LIN {X 0,Y 90.441,Z 484.223,A -85,B 0,C 180,E1 -28590.27,E2 -28590.27} C_VEL
LIN {X 0,Y 89.937,Z 477.189,A -85,B 0,C 180,E1 -28595.779,E2 -28595.779} C_VEL
LIN {X 0,Y 88.998,Z 470.496,A -85,B 0,C 180,E1 -28601.586,E2 -28601.586} C_VEL
LIN {X 0,Y 88.423,Z 466.907,A -85,B 0,C 180,E1 -28605.03,E2 -28605.03} C_VEL
LIN {X 0,Y 87.757,Z 463.816,A -85,B 0,C 180,E1 -28608.45,E2 -28608.45} C_VEL
LIN {X 0,Y 86.788,Z 460.611,A -85,B 0,C 180,E1 -28613.023,E2 -28613.023} C_VEL
LIN {X 0,Y 85.348,Z 457.502,A -85,B 0,C 180,E1 -28620,E2 -28620} C_VEL
LIN {X 0,Y 84.954,Z 455.593,A -85,B 0,C 180,E1 -28624.745,E2 -28624.745} C_VEL
LIN {X 0,Y 84.227,Z 455.367,A -85,B 0,C 180,E1 -28634.496,E2 -28634.496} C_VEL
LIN {X 0,Y 84.372,Z 456.038,A -85,B 0,C 180,E1 -28639.462,E2 -28639.462} C_VEL
LIN {X 0,Y 85.474,Z 459.487,A -85,B 0,C 180,E1 -28649.56,E2 -28649.56} C_VEL
LIN {X 0,Y 87.06,Z 463.676,A -85,B 0,C 180,E1 -28657.257,E2 -28657.257} C_VEL
LIN {X 0,Y 88.372,Z 467.412,A -85,B 0,C 180,E1 -28662.533,E2 -28662.533} C_VEL
LIN {X 0,Y 89.775,Z 472.169,A -85,B 0,C 180,E1 -28668.124,E2 -28668.124} C_VEL
LIN {X 0,Y 90.788,Z 476.909,A -85,B 0,C 180,E1 -28672.909,E2 -28672.909} C_VEL
LIN {X 0,Y 91.718,Z 483.277,A -85,B 0,C 180,E1 -28678.72,E2 -28678.72} C_VEL
LIN {X 0,Y 91.813,Z 484.853,A -85,B 0,C 180,E1 -28680.112,E2 -28680.112} C_VEL
LIN {X 0,Y 91.514,Z 486.512,A -85,B 0,C 180,E1 -28681.287,E2 -28681.287} C_VEL
LIN {X 0,Y 85.387,Z 495.474,A -85,B 0,C 180,E1 -28685.689,E2 -28685.689} C_VEL
LIN {X 0,Y 78.734,Z 504.116,A -85,B 0,C 180,E1 -28691.785,E2 -28691.785} C_VEL
LIN {X 0,Y 73.023,Z 511.07,A -85,B 0,C 180,E1 -28698.891,E2 -28698.891} C_VEL
LIN {X 0,Y 68.391,Z 516.618,A -85,B 0,C 180,E1 -28707.044,E2 -28707.044} C_VEL
LIN {X 0,Y 65.021,Z 520.925,A -85,B 0,C 180,E1 -28716.193,E2 -28716.193} C_VEL
LIN {X 0,Y 63.992,Z 522.397,A -85,B 0,C 180,E1 -28720.372,E2 -28720.372} C_VEL
LIN {X 0,Y 62.488,Z 523.952,A -85,B 0,C 180,E1 -28725.374,E2 -28725.374} C_VEL
LIN {X 0,Y 59.217,Z 525.988,A -85,B 0,C 180,E1 -28734.001,E2 -28734.001} C_VEL
LIN {X 0,Y 57.425,Z 527.14,A -85,B 0,C 180,E1 -28741.567,E2 -28741.567} C_VEL
LIN {X 0,Y 57.494,Z 527.667,A -85,B 0,C 180,E1 -28747.475,E2 -28747.475} C_VEL
LIN {X 0,Y 57.899,Z 527.754,A -85,B 0,C 180,E1 -28749.398,E2 -28749.398} C_VEL
LIN {X 0,Y 59.806,Z 527.977,A -85,B 0,C 180,E1 -28755.165,E2 -28755.165} C_VEL
LIN {X 0,Y 62.746,Z 527.792,A -85,B 0,C 180,E1 -28761.611,E2 -28761.611} C_VEL
LIN {X 0,Y 66.995,Z 527.076,A -85,B 0,C 180,E1 -28768.365,E2 -28768.365} C_VEL
LIN {X 0,Y 70.922,Z 526.057,A -85,B 0,C 180,E1 -28773.081,E2 -28773.081} C_VEL
LIN {X 0,Y 76.45,Z 524.23,A -85,B 0,C 180,E1 -28778.426,E2 -28778.426} C_VEL
LIN {X 0,Y 84.043,Z 521.069,A -85,B 0,C 180,E1 -28784.048,E2 -28784.048} C_VEL
LIN {X 0,Y 93.053,Z 516.427,A -85,B 0,C 180,E1 -28789.016,E2 -28789.016} C_VEL
LIN {X 0,Y 102.281,Z 510.549,A -85,B 0,C 180,E1 -28793.037,E2 -28793.037} C_VEL
LIN {X 0,Y 103.385,Z 509.573,A -85,B 0,C 180,E1 -28794.148,E2 -28794.148} C_VEL
LIN {X 0,Y 104.857,Z 507.368,A -85,B 0,C 180,E1 -28800,E2 -28800} C_VEL
LIN {X 0,Y 105.694,Z 506.321,A -85,B 0,C 180,E1 -28804.242,E2 -28804.242} C_VEL
LIN {X 0,Y 105.435,Z 506.439,A -85,B 0,C 180,E1 -28807.662,E2 -28807.662} C_VEL
LIN {X 0,Y 104.952,Z 507.069,A -85,B 0,C 180,E1 -28811.589,E2 -28811.589} C_VEL
LIN {X 0,Y 104.419,Z 508.123,A -85,B 0,C 180,E1 -28815.618,E2 -28815.618} C_VEL
LIN {X 0,Y 103.533,Z 509.855,A -85,B 0,C 180,E1 -28819.841,E2 -28819.841} C_VEL
LIN {X 0,Y 101.953,Z 512.493,A -85,B 0,C 180,E1 -28824.432,E2 -28824.432} C_VEL
LIN {X 0,Y 101.315,Z 513.342,A -85,B 0,C 180,E1 -28825.627,E2 -28825.627} C_VEL
LIN {X 0,Y 96.268,Z 517.412,A -85,B 0,C 180,E1 -28828.849,E2 -28828.849} C_VEL
LIN {X 0,Y 87.845,Z 522.625,A -85,B 0,C 180,E1 -28832.873,E2 -28832.873} C_VEL
LIN {X 0,Y 79.912,Z 526.75,A -85,B 0,C 180,E1 -28837.689,E2 -28837.689} C_VEL
LIN {X 0,Y 75.036,Z 528.969,A -85,B 0,C 180,E1 -28841.487,E2 -28841.487} C_VEL
LIN {X 0,Y 66.422,Z 532.14,A -85,B 0,C 180,E1 -28850.607,E2 -28850.607} C_VEL
LIN {X 0,Y 59.941,Z 533.826,A -85,B 0,C 180,E1 -28862.046,E2 -28862.046} C_VEL
LIN {X 0,Y 56.515,Z 533.981,A -85,B 0,C 180,E1 -28875.613,E2 -28875.613} C_VEL
LIN {X 0,Y 55.964,Z 533.494,A -85,B 0,C 180,E1 -28882.8,E2 -28882.8} C_VEL
LIN {X 0,Y 56.103,Z 532.623,A -85,B 0,C 180,E1 -28890.014,E2 -28890.014} C_VEL
LIN {X 0,Y 56.014,Z 531.262,A -85,B 0,C 180,E1 -28897.222,E2 -28897.222} C_VEL
LIN {X 0,Y 57.203,Z 528.349,A -85,B 0,C 180,E1 -28907.902,E2 -28907.902} C_VEL
LIN {X 0,Y 60.084,Z 524.365,A -85,B 0,C 180,E1 -28917.91,E2 -28917.91} C_VEL
LIN {X 0,Y 65.45,Z 518.205,A -85,B 0,C 180,E1 -28928.143,E2 -28928.143} C_VEL
LIN {X 0,Y 71.779,Z 510.926,A -85,B 0,C 180,E1 -28936.081,E2 -28936.081} C_VEL
LIN {X 0,Y 77.139,Z 504.599,A -85,B 0,C 180,E1 -28940.762,E2 -28940.762} C_VEL
LIN {X 0,Y 80.643,Z 497.54,A -85,B 0,C 180,E1 -28945.901,E2 -28945.901} C_VEL
LIN {X 0,Y 84.079,Z 489.495,A -85,B 0,C 180,E1 -28950.853,E2 -28950.853} C_VEL
LIN {X 0,Y 84.644,Z 487.711,A -85,B 0,C 180,E1 -28951.95,E2 -28951.95} C_VEL
LIN {X 0,Y 84.762,Z 482.126,A -85,B 0,C 180,E1 -28956.675,E2 -28956.675} C_VEL
LIN {X 0,Y 84.327,Z 475.376,A -85,B 0,C 180,E1 -28963.04,E2 -28963.04} C_VEL
LIN {X 0,Y 84.038,Z 471.877,A -85,B 0,C 180,E1 -28966.704,E2 -28966.704} C_VEL
LIN {X 0,Y 83.62,Z 468.911,A -85,B 0,C 180,E1 -28970.323,E2 -28970.323} C_VEL
LIN {X 0,Y 82.89,Z 465.961,A -85,B 0,C 180,E1 -28975.136,E2 -28975.136} C_VEL
LIN {X 0,Y 81.806,Z 462.103,A -85,B 0,C 180,E1 -28984.928,E2 -28984.928} C_VEL
LIN {X 0,Y 81.308,Z 461.735,A -85,B 0,C 180,E1 -28989.955,E2 -28989.955} C_VEL
LIN {X 0,Y 81.14,Z 461.858,A -85,B 0,C 180,E1 -28995.061,E2 -28995.061} C_VEL
LIN {X 0,Y 81.15,Z 462.183,A -85,B 0,C 180,E1 -28997.675,E2 -28997.675} C_VEL
LIN {X 0,Y 81.373,Z 464.57,A -85,B 0,C 180,E1 -29005.584,E2 -29005.584} C_VEL
LIN {X 0,Y 82.082,Z 466.661,A -85,B 0,C 180,E1 -29011.089,E2 -29011.089} C_VEL
LIN {X 0,Y 82.948,Z 469.361,A -85,B 0,C 180,E1 -29016.377,E2 -29016.377} C_VEL
LIN {X 0,Y 84.19,Z 474.136,A -85,B 0,C 180,E1 -29023.498,E2 -29023.498} C_VEL
LIN {X 0,Y 85.05,Z 478.302,A -85,B 0,C 180,E1 -29028.607,E2 -29028.607} C_VEL
LIN {X 0,Y 85.741,Z 484.381,A -85,B 0,C 180,E1 -29035.052,E2 -29035.052} C_VEL
LIN {X 0,Y 85.877,Z 486.915,A -85,B 0,C 180,E1 -29037.587,E2 -29037.587} C_VEL
LIN {X 0,Y 85.271,Z 488.72,A -85,B 0,C 180,E1 -29038.852,E2 -29038.852} C_VEL
LIN {X 0,Y 78.274,Z 498.056,A -85,B 0,C 180,E1 -29043.879,E2 -29043.879} C_VEL
LIN {X 0,Y 71.751,Z 505.832,A -85,B 0,C 180,E1 -29049.94,E2 -29049.94} C_VEL
LIN {X 0,Y 65.785,Z 512.512,A -85,B 0,C 180,E1 -29057.651,E2 -29057.651} C_VEL
LIN {X 0,Y 60.935,Z 517.82,A -85,B 0,C 180,E1 -29066.681,E2 -29066.681} C_VEL
LIN {X 0,Y 57.053,Z 522.583,A -85,B 0,C 180,E1 -29079.022,E2 -29079.022} C_VEL
LIN {X 0,Y 55.679,Z 525.751,A -85,B 0,C 180,E1 -29092.236,E2 -29092.236} C_VEL
LIN {X 0,Y 56.136,Z 526.928,A -85,B 0,C 180,E1 -29100.035,E2 -29100.035} C_VEL
LIN {X 0,Y 57.899,Z 527.754,A -85,B 0,C 180,E1 -29109.398,E2 -29109.398} C_VEL
LIN {X 0,Y 59.042,Z 528.024,A -85,B 0,C 180,E1 -29115.071,E2 -29115.071} C_VEL
LIN {X 0,Y 60.377,Z 527.97,A -85,B 0,C 180,E1 -29124.505,E2 -29124.505} C_VEL
LIN {X 0,Y 62.37,Z 527.54,A -85,B 0,C 180,E1 -29131.69,E2 -29131.69} C_VEL
LIN {X 0,Y 65.1,Z 526.861,A -85,B 0,C 180,E1 -29136.377,E2 -29136.377} C_VEL
LIN {X 0,Y 66.308,Z 526.494,A -85,B 0,C 180,E1 -29137.716,E2 -29137.716} C_VEL
LIN {X 0,Y 76.139,Z 523.39,A -85,B 0,C 180,E1 -29145.696,E2 -29145.696} C_VEL
LIN {X 0,Y 85.388,Z 519.424,A -85,B 0,C 180,E1 -29150.934,E2 -29150.934} C_VEL
LIN {X 0,Y 94.427,Z 514.574,A -85,B 0,C 180,E1 -29154.868,E2 -29154.868} C_VEL
LIN {X 0,Y 97.002,Z 512.984,A -85,B 0,C 180,E1 -29155.846,E2 -29155.846} C_VEL
LIN {X 0,Y 98.399,Z 511.735,A -85,B 0,C 180,E1 -29158.778,E2 -29158.778} C_VEL
LIN {X 0,Y 99.81,Z 510.338,A -85,B 0,C 180,E1 -29164.038,E2 -29164.038} C_VEL
LIN {X 0,Y 99.426,Z 510.581,A -85,B 0,C 180,E1 -29168.334,E2 -29168.334} C_VEL
LIN {X 0,Y 98.88,Z 511.281,A -85,B 0,C 180,E1 -29172.312,E2 -29172.312} C_VEL
LIN {X 0,Y 98.084,Z 512.526,A -85,B 0,C 180,E1 -29176.656,E2 -29176.656} C_VEL
LIN {X 0,Y 96.683,Z 514.564,A -85,B 0,C 180,E1 -29181.313,E2 -29181.313} C_VEL
LIN {X 0,Y 95.153,Z 516.094,A -85,B 0,C 180,E1 -29183.597,E2 -29183.597} C_VEL
LIN {X 0,Y 90.116,Z 519.454,A -85,B 0,C 180,E1 -29186.273,E2 -29186.273} C_VEL
LIN {X 0,Y 81.309,Z 524.147,A -85,B 0,C 180,E1 -29190.212,E2 -29190.212} C_VEL
LIN {X 0,Y 72.777,Z 527.943,A -85,B 0,C 180,E1 -29195.41,E2 -29195.41} C_VEL
LIN {X 0,Y 65.575,Z 530.553,A -85,B 0,C 180,E1 -29201.409,E2 -29201.409} C_VEL
LIN {X 0,Y 57.067,Z 532.862,A -85,B 0,C 180,E1 -29212.01,E2 -29212.01} C_VEL
LIN {X 0,Y 51.27,Z 533.634,A -85,B 0,C 180,E1 -29225.735,E2 -29225.735} C_VEL
LIN {X 0,Y 48.918,Z 532.935,A -85,B 0,C 180,E1 -29241.756,E2 -29241.756} C_VEL
LIN {X 0,Y 49.001,Z 532.012,A -85,B 0,C 180,E1 -29250.016,E2 -29250.016} C_VEL
LIN {X 0,Y 48.962,Z 530.551,A -85,B 0,C 180,E1 -29258.268,E2 -29258.268} C_VEL
LIN {X 0,Y 50.484,Z 527.539,A -85,B 0,C 180,E1 -29270.383,E2 -29270.383} C_VEL
LIN {X 0,Y 53.89,Z 523.437,A -85,B 0,C 180,E1 -29281.459,E2 -29281.459} C_VEL
LIN {X 0,Y 59.997,Z 517.137,A -85,B 0,C 180,E1 -29292.358,E2 -29292.358} C_VEL
LIN {X 0,Y 66.782,Z 509.967,A -85,B 0,C 180,E1 -29300.253,E2 -29300.253} C_VEL
LIN {X 0,Y 71.53,Z 504.715,A -85,B 0,C 180,E1 -29304.17,E2 -29304.17} C_VEL
LIN {X 0,Y 75.432,Z 497.757,A -85,B 0,C 180,E1 -29309.54,E2 -29309.54} C_VEL
LIN {X 0,Y 78.485,Z 491.588,A -85,B 0,C 180,E1 -29313.587,E2 -29313.587} C_VEL
LIN {X 0,Y 79.11,Z 489.992,A -85,B 0,C 180,E1 -29314.678,E2 -29314.678} C_VEL
LIN {X 0,Y 79.448,Z 483.823,A -85,B 0,C 180,E1 -29320.626,E2 -29320.626} C_VEL
LIN {X 0,Y 79.489,Z 478.327,A -85,B 0,C 180,E1 -29326.583,E2 -29326.583} C_VEL
LIN {X 0,Y 79.317,Z 473.834,A -85,B 0,C 180,E1 -29332.362,E2 -29332.362} C_VEL
LIN {X 0,Y 79.094,Z 472.344,A -85,B 0,C 180,E1 -29334.902,E2 -29334.902} C_VEL
LIN {X 0,Y 78.327,Z 468.39,A -85,B 0,C 180,E1 -29345.147,E2 -29345.147} C_VEL
LIN {X 0,Y 77.89,Z 467.98,A -85,B 0,C 180,E1 -29350.396,E2 -29350.396} C_VEL
LIN {X 0,Y 77.71,Z 468.178,A -85,B 0,C 180,E1 -29355.742,E2 -29355.742} C_VEL
LIN {X 0,Y 77.625,Z 470.599,A -85,B 0,C 180,E1 -29365.104,E2 -29365.104} C_VEL
LIN {X 0,Y 78.239,Z 473.491,A -85,B 0,C 180,E1 -29372.613,E2 -29372.613} C_VEL
LIN {X 0,Y 78.927,Z 476.658,A -85,B 0,C 180,E1 -29378.558,E2 -29378.558} C_VEL
LIN {X 0,Y 79.612,Z 480.989,A -85,B 0,C 180,E1 -29385.059,E2 -29385.059} C_VEL
LIN {X 0,Y 79.935,Z 485.011,A -85,B 0,C 180,E1 -29390.085,E2 -29390.085} C_VEL
LIN {X 0,Y 80.042,Z 489.079,A -85,B 0,C 180,E1 -29394.822,E2 -29394.822} C_VEL
LIN {X 0,Y 79.105,Z 490.913,A -85,B 0,C 180,E1 -29396.076,E2 -29396.076} C_VEL
LIN {X 0,Y 72.231,Z 499.397,A -85,B 0,C 180,E1 -29400.878,E2 -29400.878} C_VEL
LIN {X 0,Y 64.894,Z 507.442,A -85,B 0,C 180,E1 -29407.713,E2 -29407.713} C_VEL
LIN {X 0,Y 58.526,Z 513.89,A -85,B 0,C 180,E1 -29416.09,E2 -29416.09} C_VEL
LIN {X 0,Y 53.476,Z 519.006,A -85,B 0,C 180,E1 -29426.218,E2 -29426.218} C_VEL
LIN {X 0,Y 49.813,Z 523.223,A -85,B 0,C 180,E1 -29439.028,E2 -29439.028} C_VEL
LIN {X 0,Y 48.789,Z 524.988,A -85,B 0,C 180,E1 -29446.727,E2 -29446.727} C_VEL
LIN {X 0,Y 49.083,Z 527.2,A -85,B 0,C 180,E1 -29460.784,E2 -29460.784} C_VEL
LIN {X 0,Y 51.529,Z 528.252,A -85,B 0,C 180,E1 -29472.974,E2 -29472.974} C_VEL
LIN {X 0,Y 54.458,Z 528.412,A -85,B 0,C 180,E1 -29480.72,E2 -29480.72} C_VEL
LIN {X 0,Y 58.189,Z 528.147,A -85,B 0,C 180,E1 -29487.693,E2 -29487.693} C_VEL
LIN {X 0,Y 62.669,Z 527.402,A -85,B 0,C 180,E1 -29493.757,E2 -29493.757} C_VEL
LIN {X 0,Y 66.308,Z 526.494,A -85,B 0,C 180,E1 -29497.716,E2 -29497.716} C_VEL
LIN {X 0,Y 69.792,Z 525.541,A -85,B 0,C 180,E1 -29501.66,E2 -29501.66} C_VEL
LIN {X 0,Y 74.846,Z 523.681,A -85,B 0,C 180,E1 -29508.271,E2 -29508.271} C_VEL
LIN {X 0,Y 80.569,Z 521.096,A -85,B 0,C 180,E1 -29513.925,E2 -29513.925} C_VEL
LIN {X 0,Y 84.857,Z 519.007,A -85,B 0,C 180,E1 -29516.331,E2 -29516.331} C_VEL
LIN {X 0,Y 91.37,Z 515.634,A -85,B 0,C 180,E1 -29518.767,E2 -29518.767} C_VEL
LIN {X 0,Y 92.402,Z 514.992,A -85,B 0,C 180,E1 -29520,E2 -29520} C_VEL
LIN {X 0,Y 93.655,Z 514.058,A -85,B 0,C 180,E1 -29524.304,E2 -29524.304} C_VEL
LIN {X 0,Y 93.23,Z 514.366,A -85,B 0,C 180,E1 -29528.672,E2 -29528.672} C_VEL
LIN {X 0,Y 92.462,Z 515.24,A -85,B 0,C 180,E1 -29533.181,E2 -29533.181} C_VEL
LIN {X 0,Y 91.316,Z 516.685,A -85,B 0,C 180,E1 -29537.93,E2 -29537.93} C_VEL
LIN {X 0,Y 90.045,Z 517.894,A -85,B 0,C 180,E1 -29540.539,E2 -29540.539} C_VEL
LIN {X 0,Y 87.167,Z 519.66,A -85,B 0,C 180,E1 -29542.024,E2 -29542.024} C_VEL
LIN {X 0,Y 77.972,Z 524.22,A -85,B 0,C 180,E1 -29545.689,E2 -29545.689} C_VEL
LIN {X 0,Y 66.437,Z 528.712,A -85,B 0,C 180,E1 -29552.215,E2 -29552.215} C_VEL
LIN {X 0,Y 56.114,Z 531.645,A -85,B 0,C 180,E1 -29561.304,E2 -29561.304} C_VEL
LIN {X 0,Y 47.795,Z 533.023,A -85,B 0,C 180,E1 -29573.993,E2 -29573.993} C_VEL
LIN {X 0,Y 42.863,Z 532.952,A -85,B 0,C 180,E1 -29590.877,E2 -29590.877} C_VEL
LIN {X 0,Y 41.913,Z 532.367,A -85,B 0,C 180,E1 -29600.366,E2 -29600.366} C_VEL
LIN {X 0,Y 41.909,Z 531.355,A -85,B 0,C 180,E1 -29610.018,E2 -29610.018} C_VEL
LIN {X 0,Y 41.954,Z 529.828,A -85,B 0,C 180,E1 -29619.662,E2 -29619.662} C_VEL
LIN {X 0,Y 43.864,Z 526.7,A -85,B 0,C 180,E1 -29633.632,E2 -29633.632} C_VEL
LIN {X 0,Y 47.938,Z 522.479,A -85,B 0,C 180,E1 -29645.923,E2 -29645.923} C_VEL
LIN {X 0,Y 54.937,Z 516.055,A -85,B 0,C 180,E1 -29657.377,E2 -29657.377} C_VEL
LIN {X 0,Y 62.198,Z 508.957,A -85,B 0,C 180,E1 -29665.066,E2 -29665.066} C_VEL
LIN {X 0,Y 66.212,Z 504.813,A -85,B 0,C 180,E1 -29668.14,E2 -29668.14} C_VEL
LIN {X 0,Y 70.548,Z 497.906,A -85,B 0,C 180,E1 -29673.734,E2 -29673.734} C_VEL
LIN {X 0,Y 73.544,Z 492.433,A -85,B 0,C 180,E1 -29677.527,E2 -29677.527} C_VEL
LIN {X 0,Y 74.259,Z 486.999,A -85,B 0,C 180,E1 -29683.505,E2 -29683.505} C_VEL
LIN {X 0,Y 74.712,Z 482.326,A -85,B 0,C 180,E1 -29689.155,E2 -29689.155} C_VEL
LIN {X 0,Y 74.871,Z 478.616,A -85,B 0,C 180,E1 -29694.613,E2 -29694.613} C_VEL
LIN {X 0,Y 74.578,Z 476.29,A -85,B 0,C 180,E1 -29700,E2 -29700} C_VEL
LIN {X 0,Y 74.428,Z 474.435,A -85,B 0,C 180,E1 -29705.955,E2 -29705.955} C_VEL
LIN {X 0,Y 74.119,Z 474.05,A -85,B 0,C 180,E1 -29710.931,E2 -29710.931} C_VEL
LIN {X 0,Y 73.723,Z 474.655,A -85,B 0,C 180,E1 -29717.549,E2 -29717.549} C_VEL
LIN {X 0,Y 73.548,Z 475.826,A -85,B 0,C 180,E1 -29722.471,E2 -29722.471} C_VEL
LIN {X 0,Y 73.794,Z 478.622,A -85,B 0,C 180,E1 -29730.984,E2 -29730.984} C_VEL
LIN {X 0,Y 74.109,Z 481.26,A -85,B 0,C 180,E1 -29736.587,E2 -29736.587} C_VEL
LIN {X 0,Y 74.396,Z 485.323,A -85,B 0,C 180,E1 -29743.47,E2 -29743.47} C_VEL
LIN {X 0,Y 74.358,Z 489.359,A -85,B 0,C 180,E1 -29749.123,E2 -29749.123} C_VEL
LIN {X 0,Y 74.27,Z 491.359,A -85,B 0,C 180,E1 -29751.771,E2 -29751.771} C_VEL
LIN {X 0,Y 73.025,Z 493.187,A -85,B 0,C 180,E1 -29752.88,E2 -29752.88} C_VEL
LIN {X 0,Y 65.9,Z 501.232,A -85,B 0,C 180,E1 -29757.763,E2 -29757.763} C_VEL
LIN {X 0,Y 58.105,Z 509.001,A -85,B 0,C 180,E1 -29764.94,E2 -29764.94} C_VEL
LIN {X 0,Y 51.021,Z 515.533,A -85,B 0,C 180,E1 -29774.628,E2 -29774.628} C_VEL
LIN {X 0,Y 45.965,Z 520.168,A -85,B 0,C 180,E1 -29785.599,E2 -29785.599} C_VEL
LIN {X 0,Y 42.483,Z 523.933,A -85,B 0,C 180,E1 -29799.504,E2 -29799.504} C_VEL
LIN {X 0,Y 41.545,Z 525.813,A -85,B 0,C 180,E1 -29809.755,E2 -29809.755} C_VEL
LIN {X 0,Y 42.27,Z 527.651,A -85,B 0,C 180,E1 -29823.767,E2 -29823.767} C_VEL
LIN {X 0,Y 46.144,Z 528.766,A -85,B 0,C 180,E1 -29839.572,E2 -29839.572} C_VEL
LIN {X 0,Y 49.867,Z 528.849,A -85,B 0,C 180,E1 -29847.706,E2 -29847.706} C_VEL
LIN {X 0,Y 57.68,Z 527.984,A -85,B 0,C 180,E1 -29858.56,E2 -29858.56} C_VEL
LIN {X 0,Y 65.306,Z 526.283,A -85,B 0,C 180,E1 -29865.539,E2 -29865.539} C_VEL
LIN {X 0,Y 74.584,Z 523.35,A -85,B 0,C 180,E1 -29871.576,E2 -29871.576} C_VEL
LIN {X 0,Y 84.857,Z 519.007,A -85,B 0,C 180,E1 -29876.331,E2 -29876.331} C_VEL
LIN {X 0,Y 86.147,Z 518.315,A -85,B 0,C 180,E1 -29877.489,E2 -29877.489} C_VEL
LIN {X 0,Y 86.682,Z 517.932,A -85,B 0,C 180,E1 -29879.492,E2 -29879.492} C_VEL
LIN {X 0,Y 86.971,Z 517.633,A -85,B 0,C 180,E1 -29883.597,E2 -29883.597} C_VEL
LIN {X 0,Y 87.316,Z 517.45,A -85,B 0,C 180,E1 -29884.617,E2 -29884.617} C_VEL
LIN {X 0,Y 86.809,Z 517.845,A -85,B 0,C 180,E1 -29889.319,E2 -29889.319} C_VEL
LIN {X 0,Y 86.268,Z 518.381,A -85,B 0,C 180,E1 -29892.195,E2 -29892.195} C_VEL
LIN {X 0,Y 85.66,Z 518.923,A -85,B 0,C 180,E1 -29894.249,E2 -29894.249} C_VEL
LIN {X 0,Y 84.135,Z 520.127,A -85,B 0,C 180,E1 -29897.684,E2 -29897.684} C_VEL
LIN {X 0,Y 72.028,Z 525.5,A -85,B 0,C 180,E1 -29902.068,E2 -29902.068} C_VEL
LIN {X 0,Y 62.918,Z 528.601,A -85,B 0,C 180,E1 -29906.7,E2 -29906.7} C_VEL
LIN {X 0,Y 57.16,Z 530.193,A -85,B 0,C 180,E1 -29910.637,E2 -29910.637} C_VEL
LIN {X 0,Y 46.662,Z 532.173,A -85,B 0,C 180,E1 -29921.169,E2 -29921.169} C_VEL
LIN {X 0,Y 38.696,Z 532.705,A -85,B 0,C 180,E1 -29937.009,E2 -29937.009} C_VEL
LIN {X 0,Y 36.201,Z 532.434,A -85,B 0,C 180,E1 -29947.176,E2 -29947.176} C_VEL
LIN {X 0,Y 34.923,Z 531.758,A -85,B 0,C 180,E1 -29958.413,E2 -29958.413} C_VEL
LIN {X 0,Y 34.809,Z 530.675,A -85,B 0,C 180,E1 -29970.022,E2 -29970.022} C_VEL
LIN {X 0,Y 35.487,Z 528.129,A -85,B 0,C 180,E1 -29987.304,E2 -29987.304} C_VEL
LIN {X 0,Y 38.856,Z 524.529,A -85,B 0,C 180,E1 -30002.885,E2 -30002.885} C_VEL
LIN {X 0,Y 44.456,Z 519.789,A -85,B 0,C 180,E1 -30015.373,E2 -30015.373} C_VEL
LIN {X 0,Y 51.626,Z 513.774,A -85,B 0,C 180,E1 -30024.79,E2 -30024.79} C_VEL
LIN {X 0,Y 59.291,Z 506.786,A -85,B 0,C 180,E1 -30031.407,E2 -30031.407} C_VEL
LIN {X 0,Y 61.107,Z 505.056,A -85,B 0,C 180,E1 -30032.609,E2 -30032.609} C_VEL
LIN {X 0,Y 66.092,Z 498,A -85,B 0,C 180,E1 -30038.534,E2 -30038.534} C_VEL
LIN {X 0,Y 68.163,Z 494.616,A -85,B 0,C 180,E1 -30041.081,E2 -30041.081} C_VEL
LIN {X 0,Y 69.408,Z 488.894,A -85,B 0,C 180,E1 -30048.316,E2 -30048.316} C_VEL
LIN {X 0,Y 69.809,Z 486.699,A -85,B 0,C 180,E1 -30051.314,E2 -30051.314} C_VEL
LIN {X 0,Y 70.294,Z 483.263,A -85,B 0,C 180,E1 -30057.134,E2 -30057.134} C_VEL
LIN {X 0,Y 70.273,Z 482.107,A -85,B 0,C 180,E1 -30060,E2 -30060} C_VEL
LIN {X 0,Y 70.297,Z 480.313,A -85,B 0,C 180,E1 -30065.737,E2 -30065.737} C_VEL
LIN {X 0,Y 69.944,Z 479.931,A -85,B 0,C 180,E1 -30071.593,E2 -30071.593} C_VEL
LIN {X 0,Y 69.511,Z 480.542,A -85,B 0,C 180,E1 -30077.657,E2 -30077.657} C_VEL
LIN {X 0,Y 69.187,Z 482.955,A -85,B 0,C 180,E1 -30087.2,E2 -30087.2} C_VEL
LIN {X 0,Y 69.179,Z 485.236,A -85,B 0,C 180,E1 -30093.308,E2 -30093.308} C_VEL
LIN {X 0,Y 69.173,Z 487.212,A -85,B 0,C 180,E1 -30097.56,E2 -30097.56} C_VEL
LIN {X 0,Y 68.968,Z 491.137,A -85,B 0,C 180,E1 -30104.48,E2 -30104.48} C_VEL
LIN {X 0,Y 68.643,Z 493.705,A -85,B 0,C 180,E1 -30108.35,E2 -30108.35} C_VEL
LIN {X 0,Y 59.774,Z 502.984,A -85,B 0,C 180,E1 -30113.978,E2 -30113.978} C_VEL
LIN {X 0,Y 51.509,Z 510.52,A -85,B 0,C 180,E1 -30121.458,E2 -30121.458} C_VEL
LIN {X 0,Y 44.214,Z 516.518,A -85,B 0,C 180,E1 -30131.445,E2 -30131.445} C_VEL
LIN {X 0,Y 38.463,Z 521.246,A -85,B 0,C 180,E1 -30144.738,E2 -30144.738} C_VEL
LIN {X 0,Y 34.975,Z 524.844,A -85,B 0,C 180,E1 -30161.57,E2 -30161.57} C_VEL
LIN {X 0,Y 34.415,Z 526.644,A -85,B 0,C 180,E1 -30174.081,E2 -30174.081} C_VEL
LIN {X 0,Y 35.61,Z 528.098,A -85,B 0,C 180,E1 -30187.868,E2 -30187.868} C_VEL
LIN {X 0,Y 41.514,Z 529.28,A -85,B 0,C 180,E1 -30207.792,E2 -30207.792} C_VEL
LIN {X 0,Y 46.153,Z 529.266,A -85,B 0,C 180,E1 -30215.973,E2 -30215.973} C_VEL
LIN {X 0,Y 53.809,Z 528.458,A -85,B 0,C 180,E1 -30224.858,E2 -30224.858} C_VEL
LIN {X 0,Y 66.319,Z 525.668,A -85,B 0,C 180,E1 -30233.917,E2 -30233.917} C_VEL
LIN {X 0,Y 77.304,Z 521.962,A -85,B 0,C 180,E1 -30239.044,E2 -30239.044} C_VEL
LIN {X 0,Y 84.351,Z 518.898,A -85,B 0,C 180,E1 -30241.541,E2 -30241.541} C_VEL
LIN {X 0,Y 86.804,Z 517.728,A -85,B 0,C 180,E1 -30243.07,E2 -30243.07} C_VEL
LIN {X 0,Y 86.971,Z 517.633,A -85,B 0,C 180,E1 -30243.597,E2 -30243.597} C_VEL
LIN {X 0,Y 87.021,Z 517.607,A -85,B 0,C 180,E1 -30245.355,E2 -30245.355} C_VEL
LIN {X 0,Y 86.329,Z 517.988,A -85,B 0,C 180,E1 -30247.073,E2 -30247.073} C_VEL
LIN {X 0,Y 84.385,Z 519.026,A -85,B 0,C 180,E1 -30249.488,E2 -30249.488} C_VEL
LIN {X 0,Y 80.558,Z 521.018,A -85,B 0,C 180,E1 -30252.381,E2 -30252.381} C_VEL
LIN {X 0,Y 77.088,Z 522.611,A -85,B 0,C 180,E1 -30254.192,E2 -30254.192} C_VEL
LIN {X 0,Y 74.512,Z 523.672,A -85,B 0,C 180,E1 -30255.11,E2 -30255.11} C_VEL
LIN {X 0,Y 66.428,Z 526.591,A -85,B 0,C 180,E1 -30257.832,E2 -30257.832} C_VEL
LIN {X 0,Y 60.048,Z 528.493,A -85,B 0,C 180,E1 -30260.597,E2 -30260.597} C_VEL
LIN {X 0,Y 47.904,Z 531.079,A -85,B 0,C 180,E1 -30268.362,E2 -30268.362} C_VEL
LIN {X 0,Y 37.207,Z 532.208,A -85,B 0,C 180,E1 -30280.958,E2 -30280.958} C_VEL
LIN {X 0,Y 29.766,Z 531.868,A -85,B 0,C 180,E1 -30301.852,E2 -30301.852} C_VEL
LIN {X 0,Y 28.009,Z 531.127,A -85,B 0,C 180,E1 -30315.497,E2 -30315.497} C_VEL
LIN {X 0,Y 27.722,Z 529.993,A -85,B 0,C 180,E1 -30330.028,E2 -30330.028} C_VEL
LIN {X 0,Y 28.766,Z 527.329,A -85,B 0,C 180,E1 -30351.527,E2 -30351.527} C_VEL
LIN {X 0,Y 33.093,Z 523.608,A -85,B 0,C 180,E1 -30369.606,E2 -30369.606} C_VEL
LIN {X 0,Y 39.778,Z 518.742,A -85,B 0,C 180,E1 -30382.692,E2 -30382.692} C_VEL
LIN {X 0,Y 47.859,Z 512.58,A -85,B 0,C 180,E1 -30391.807,E2 -30391.807} C_VEL
LIN {X 0,Y 56.747,Z 504.922,A -85,B 0,C 180,E1 -30398.189,E2 -30398.189} C_VEL
LIN {X 0,Y 62.887,Z 497.036,A -85,B 0,C 180,E1 -30404.767,E2 -30404.767} C_VEL
LIN {X 0,Y 64.507,Z 491.929,A -85,B 0,C 180,E1 -30412.127,E2 -30412.127} C_VEL
LIN {X 0,Y 65.313,Z 489.135,A -85,B 0,C 180,E1 -30416.915,E2 -30416.915} C_VEL
LIN {X 0,Y 65.591,Z 487.755,A -85,B 0,C 180,E1 -30419.999,E2 -30419.999} C_VEL
LIN {X 0,Y 65.79,Z 485.903,A -85,B 0,C 180,E1 -30426.132,E2 -30426.132} C_VEL
LIN {X 0,Y 65.415,Z 485.634,A -85,B 0,C 180,E1 -30432.408,E2 -30432.408} C_VEL
LIN {X 0,Y 64.84,Z 486.477,A -85,B 0,C 180,E1 -30438.975,E2 -30438.975} C_VEL
LIN {X 0,Y 64.458,Z 488.038,A -85,B 0,C 180,E1 -30445.856,E2 -30445.856} C_VEL
LIN {X 0,Y 64.131,Z 490.558,A -85,B 0,C 180,E1 -30453.225,E2 -30453.225} C_VEL
LIN {X 0,Y 63.736,Z 493.37,A -85,B 0,C 180,E1 -30459.46,E2 -30459.46} C_VEL
LIN {X 0,Y 63.527,Z 494.487,A -85,B 0,C 180,E1 -30461.588,E2 -30461.588} C_VEL
LIN {X 0,Y 62.784,Z 496.293,A -85,B 0,C 180,E1 -30464.208,E2 -30464.208} C_VEL
LIN {X 0,Y 53.979,Z 504.717,A -85,B 0,C 180,E1 -30469.366,E2 -30469.366} C_VEL
LIN {X 0,Y 45.136,Z 511.942,A -85,B 0,C 180,E1 -30476.958,E2 -30476.958} C_VEL
LIN {X 0,Y 37.227,Z 517.737,A -85,B 0,C 180,E1 -30487.795,E2 -30487.795} C_VEL
LIN {X 0,Y 30.955,Z 522.297,A -85,B 0,C 180,E1 -30503.457,E2 -30503.457} C_VEL
LIN {X 0,Y 27.538,Z 525.733,A -85,B 0,C 180,E1 -30524.757,E2 -30524.757} C_VEL
LIN {X 0,Y 27.584,Z 527.445,A -85,B 0,C 180,E1 -30540.602,E2 -30540.602} C_VEL
LIN {X 0,Y 29.558,Z 528.651,A -85,B 0,C 180,E1 -30555.465,E2 -30555.465} C_VEL
LIN {X 0,Y 33.141,Z 529.435,A -85,B 0,C 180,E1 -30567.976,E2 -30567.976} C_VEL
LIN {X 0,Y 38.365,Z 529.777,A -85,B 0,C 180,E1 -30578.508,E2 -30578.508} C_VEL
LIN {X 0,Y 43.551,Z 529.627,A -85,B 0,C 180,E1 -30585.444,E2 -30585.444} C_VEL
LIN {X 0,Y 50.723,Z 528.928,A -85,B 0,C 180,E1 -30592.036,E2 -30592.036} C_VEL
LIN {X 0,Y 56.356,Z 527.994,A -85,B 0,C 180,E1 -30595.863,E2 -30595.863} C_VEL
LIN {X 0,Y 64.275,Z 526.162,A -85,B 0,C 180,E1 -30600.001,E2 -30600.001} C_VEL
LIN {X 0,Y 73.934,Z 523.156,A -85,B 0,C 180,E1 -30603.713,E2 -30603.713} C_VEL
LIN {X 0,Y 78.593,Z 521.386,A -85,B 0,C 180,E1 -30605.131,E2 -30605.131} C_VEL
LIN {X 0,Y 80.621,Z 520.587,A -85,B 0,C 180,E1 -30606.256,E2 -30606.256} C_VEL
LIN {X 0,Y 80.092,Z 521.007,A -85,B 0,C 180,E1 -30610.108,E2 -30610.108} C_VEL
LIN {X 0,Y 79.305,Z 521.583,A -85,B 0,C 180,E1 -30612.935,E2 -30612.935} C_VEL
LIN {X 0,Y 76.25,Z 522.996,A -85,B 0,C 180,E1 -30614.626,E2 -30614.626} C_VEL
LIN {X 0,Y 74.512,Z 523.672,A -85,B 0,C 180,E1 -30615.11,E2 -30615.11} C_VEL
LIN {X 0,Y 69.091,Z 525.63,A -85,B 0,C 180,E1 -30616.223,E2 -30616.223} C_VEL
LIN {X 0,Y 59.562,Z 528.254,A -85,B 0,C 180,E1 -30617.022,E2 -30617.022} C_VEL
LIN {X 0,Y 49.921,Z 530.124,A -85,B 0,C 180,E1 -30618.29,E2 -30618.29} C_VEL
LIN {X 0,Y 44.413,Z 530.855,A -85,B 0,C 180,E1 -30620.688,E2 -30620.688} C_VEL
LIN {X 0,Y 32.972,Z 531.791,A -85,B 0,C 180,E1 -30631.551,E2 -30631.551} C_VEL
LIN {X 0,Y 23.734,Z 531.288,A -85,B 0,C 180,E1 -30653.726,E2 -30653.726} C_VEL
LIN {X 0,Y 21.207,Z 530.489,A -85,B 0,C 180,E1 -30670.685,E2 -30670.685} C_VEL
LIN {X 0,Y 20.637,Z 529.298,A -85,B 0,C 180,E1 -30690.037,E2 -30690.037} C_VEL
LIN {X 0,Y 22.303,Z 526.508,A -85,B 0,C 180,E1 -30718.247,E2 -30718.247} C_VEL
LIN {X 0,Y 27.96,Z 522.652,A -85,B 0,C 180,E1 -30738.985,E2 -30738.985} C_VEL
LIN {X 0,Y 35.914,Z 517.652,A -85,B 0,C 180,E1 -30751.757,E2 -30751.757} C_VEL
LIN {X 0,Y 44.925,Z 511.322,A -85,B 0,C 180,E1 -30759.871,E2 -30759.871} C_VEL
LIN {X 0,Y 52.902,Z 504.797,A -85,B 0,C 180,E1 -30764.591,E2 -30764.591} C_VEL
LIN {X 0,Y 57.33,Z 499.826,A -85,B 0,C 180,E1 -30768.788,E2 -30768.788} C_VEL
LIN {X 0,Y 58.059,Z 498.664,A -85,B 0,C 180,E1 -30770.204,E2 -30770.204} C_VEL
LIN {X 0,Y 59.823,Z 494.825,A -85,B 0,C 180,E1 -30776.632,E2 -30776.632} C_VEL
LIN {X 0,Y 60.435,Z 493.237,A -85,B 0,C 180,E1 -30779.999,E2 -30779.999} C_VEL
LIN {X 0,Y 60.983,Z 491.246,A -85,B 0,C 180,E1 -30786.617,E2 -30786.617} C_VEL
LIN {X 0,Y 60.58,Z 491.084,A -85,B 0,C 180,E1 -30793.416,E2 -30793.416} C_VEL
LIN {X 0,Y 59.768,Z 492.172,A -85,B 0,C 180,E1 -30800.656,E2 -30800.656} C_VEL
LIN {X 0,Y 59.197,Z 494.025,A -85,B 0,C 180,E1 -30808.352,E2 -30808.352} C_VEL
LIN {X 0,Y 58.767,Z 495.603,A -85,B 0,C 180,E1 -30813.139,E2 -30813.139} C_VEL
LIN {X 0,Y 58.322,Z 497.179,A -85,B 0,C 180,E1 -30817.05,E2 -30817.05} C_VEL
LIN {X 0,Y 57.121,Z 498.914,A -85,B 0,C 180,E1 -30819.345,E2 -30819.345} C_VEL
LIN {X 0,Y 46.992,Z 507.58,A -85,B 0,C 180,E1 -30824.71,E2 -30824.71} C_VEL
LIN {X 0,Y 37.607,Z 514.368,A -85,B 0,C 180,E1 -30832.576,E2 -30832.576} C_VEL
LIN {X 0,Y 30.429,Z 518.938,A -85,B 0,C 180,E1 -30842.46,E2 -30842.46} C_VEL
LIN {X 0,Y 23.423,Z 523.342,A -85,B 0,C 180,E1 -30861.339,E2 -30861.339} C_VEL
LIN {X 0,Y 20.225,Z 526.618,A -85,B 0,C 180,E1 -30890.293,E2 -30890.293} C_VEL
LIN {X 0,Y 23.357,Z 528.982,A -85,B 0,C 180,E1 -30923.003,E2 -30923.003} C_VEL
LIN {X 0,Y 29.746,Z 530.017,A -85,B 0,C 180,E1 -30940.839,E2 -30940.839} C_VEL
LIN {X 0,Y 35.722,Z 530.221,A -85,B 0,C 180,E1 -30949.516,E2 -30949.516} C_VEL
LIN {X 0,Y 42.266,Z 529.996,A -85,B 0,C 180,E1 -30955.816,E2 -30955.816} C_VEL
LIN {X 0,Y 49.182,Z 529.326,A -85,B 0,C 180,E1 -30960.366,E2 -30960.366} C_VEL
LIN {X 0,Y 56.338,Z 528.14,A -85,B 0,C 180,E1 -30963.867,E2 -30963.867} C_VEL
LIN {X 0,Y 67.371,Z 525.476,A -85,B 0,C 180,E1 -30967.777,E2 -30967.777} C_VEL
LIN {X 0,Y 71.102,Z 524.345,A -85,B 0,C 180,E1 -30968.802,E2 -30968.802} C_VEL
LIN {X 0,Y 71.364,Z 524.334,A -85,B 0,C 180,E1 -30970.066,E2 -30970.066} C_VEL
LIN {X 0,Y 64.603,Z 526.561,A -85,B 0,C 180,E1 -30971.802,E2 -30971.802} C_VEL
LIN {X 0,Y 51.374,Z 529.756,A -85,B 0,C 180,E1 -30976.798,E2 -30976.798} C_VEL
LIN {X 0,Y 44.413,Z 530.855,A -85,B 0,C 180,E1 -30980.688,E2 -30980.688} C_VEL
LIN {X 0,Y 38.971,Z 531.404,A -85,B 0,C 180,E1 -30983.804,E2 -30983.804} C_VEL
LIN {X 0,Y 29.449,Z 531.559,A -85,B 0,C 180,E1 -30988.498,E2 -30988.498} C_VEL
LIN {X 0,Y 20.337,Z 530.951,A -85,B 0,C 180,E1 -30997.576,E2 -30997.576} C_VEL
LIN {X 0,Y 16.149,Z 530.239,A -85,B 0,C 180,E1 -31010.638,E2 -31010.638} C_VEL
LIN {X 0,Y 13.551,Z 528.584,A -85,B 0,C 180,E1 -31050.057,E2 -31050.057} C_VEL
LIN {X 0,Y 16.397,Z 525.682,A -85,B 0,C 180,E1 -31090.072,E2 -31090.072} C_VEL
LIN {X 0,Y 23.891,Z 521.691,A -85,B 0,C 180,E1 -31112.011,E2 -31112.011} C_VEL
LIN {X 0,Y 34.757,Z 515.527,A -85,B 0,C 180,E1 -31123.91,E2 -31123.91} C_VEL
LIN {X 0,Y 44.672,Z 508.76,A -85,B 0,C 180,E1 -31129.596,E2 -31129.596} C_VEL
LIN {X 0,Y 48.06,Z 506.162,A -85,B 0,C 180,E1 -31130.873,E2 -31130.873} C_VEL
LIN {X 0,Y 51.331,Z 503.166,A -85,B 0,C 180,E1 -31133.12,E2 -31133.12} C_VEL
LIN {X 0,Y 53.093,Z 501.325,A -85,B 0,C 180,E1 -31134.779,E2 -31134.779} C_VEL
LIN {X 0,Y 54.783,Z 498.557,A -85,B 0,C 180,E1 -31139.999,E2 -31139.999} C_VEL
LIN {X 0,Y 55.412,Z 497.258,A -85,B 0,C 180,E1 -31143.635,E2 -31143.635} C_VEL
LIN {X 0,Y 55.864,Z 496.315,A -85,B 0,C 180,E1 -31147.227,E2 -31147.227} C_VEL
LIN {X 0,Y 55.258,Z 496.391,A -85,B 0,C 180,E1 -31154.736,E2 -31154.736} C_VEL
LIN {X 0,Y 54.084,Z 498.066,A -85,B 0,C 180,E1 -31164.516,E2 -31164.516} C_VEL
LIN {X 0,Y 53.244,Z 500.043,A -85,B 0,C 180,E1 -31171.868,E2 -31171.868} C_VEL
LIN {X 0,Y 51.569,Z 501.761,A -85,B 0,C 180,E1 -31173.542,E2 -31173.542} C_VEL
LIN {X 0,Y 42.129,Z 509.12,A -85,B 0,C 180,E1 -31177.561,E2 -31177.561} C_VEL
LIN {X 0,Y 33.682,Z 514.682,A -85,B 0,C 180,E1 -31183.056,E2 -31183.056} C_VEL
LIN {X 0,Y 24.021,Z 520.093,A -85,B 0,C 180,E1 -31194.148,E2 -31194.148} C_VEL
LIN {X 0,Y 15.952,Z 524.309,A -85,B 0,C 180,E1 -31217.225,E2 -31217.225} C_VEL
LIN {X 0,Y 13.284,Z 527.424,A -85,B 0,C 180,E1 -31261.872,E2 -31261.872} C_VEL
LIN {X 0,Y 18.368,Z 529.406,A -85,B 0,C 180,E1 -31297.506,E2 -31297.506} C_VEL
LIN {X 0,Y 28.165,Z 530.535,A -85,B 0,C 180,E1 -31316.035,E2 -31316.035} C_VEL
LIN {X 0,Y 35.152,Z 530.663,A -85,B 0,C 180,E1 -31322.197,E2 -31322.197} C_VEL
LIN {X 0,Y 47.403,Z 529.876,A -85,B 0,C 180,E1 -31328.527,E2 -31328.527} C_VEL
LIN {X 0,Y 42.999,Z 530.518,A -85,B 0,C 180,E1 -31331.382,E2 -31331.382} C_VEL
LIN {X 0,Y 29.865,Z 531.326,A -85,B 0,C 180,E1 -31339.808,E2 -31339.808} C_VEL
LIN {X 0,Y 18.471,Z 530.7,A -85,B 0,C 180,E1 -31360.516,E2 -31360.516} C_VEL
LIN {X 0,Y 16.149,Z 530.239,A -85,B 0,C 180,E1 -31370.638,E2 -31370.638} C_VEL
LIN {X 0,Y 14.069,Z 529.716,A -85,B 0,C 180,E1 -31383.101,E2 -31383.101} C_VEL
LIN {X 0,Y 11.415,Z 528.51,A -85,B 0,C 180,E1 -31406.579,E2 -31406.579} C_VEL
LIN {X 0,Y 11.421,Z 525.78,A -85,B 0,C 180,E1 -31456.768,E2 -31456.768} C_VEL
LIN {X 0,Y 16.306,Z 523.03,A -85,B 0,C 180,E1 -31481.728,E2 -31481.728} C_VEL
LIN {X 0,Y 19.64,Z 521.47,A -85,B 0,C 180,E1 -31487.239,E2 -31487.239} C_VEL
LIN {X 0,Y 28.302,Z 517.236,A -85,B 0,C 180,E1 -31493.591,E2 -31493.591} C_VEL
LIN {X 0,Y 38.705,Z 511.043,A -85,B 0,C 180,E1 -31497.461,E2 -31497.461} C_VEL
LIN {X 0,Y 45.42,Z 506.268,A -85,B 0,C 180,E1 -31499.044,E2 -31499.044} C_VEL
LIN {X 0,Y 47.555,Z 504.52,A -85,B 0,C 180,E1 -31499.999,E2 -31499.999} C_VEL
LIN {X 0,Y 49.258,Z 502.751,A -85,B 0,C 180,E1 -31502.566,E2 -31502.566} C_VEL
LIN {X 0,Y 50.443,Z 501.072,A -85,B 0,C 180,E1 -31508.008,E2 -31508.008} C_VEL
LIN {X 0,Y 50.146,Z 501.093,A -85,B 0,C 180,E1 -31511.095,E2 -31511.095} C_VEL
LIN {X 0,Y 49.473,Z 501.528,A -85,B 0,C 180,E1 -31516.505,E2 -31516.505} C_VEL
LIN {X 0,Y 48.145,Z 503.194,A -85,B 0,C 180,E1 -31525.971,E2 -31525.971} C_VEL
LIN {X 0,Y 38.072,Z 510.534,A -85,B 0,C 180,E1 -31528.697,E2 -31528.697} C_VEL
LIN {X 0,Y 29.106,Z 515.93,A -85,B 0,C 180,E1 -31532.267,E2 -31532.267} C_VEL
LIN {X 0,Y 18.459,Z 521.174,A -85,B 0,C 180,E1 -31540.342,E2 -31540.342} C_VEL
LIN {X 0,Y 11.67,Z 524.031,A -85,B 0,C 180,E1 -31552.889,E2 -31552.889} C_VEL
LIN {X 0,Y 6.507,Z 526.369,A -85,B 0,C 180,E1 -31589.881,E2 -31589.881} C_VEL
LIN {X 0,Y 7.875,Z 528.22,A -85,B 0,C 180,E1 -31652.965,E2 -31652.965} C_VEL
LIN {X 0,Y 15.322,Z 529.834,A -85,B 0,C 180,E1 -31680.002,E2 -31680.002} C_VEL
LIN {X 0,Y 21.231,Z 530.564,A -85,B 0,C 180,E1 -31687.054,E2 -31687.054} C_VEL
LIN {X 0,Y 21.435,Z 530.663,A -85,B 0,C 180,E1 -31690.594,E2 -31690.594} C_VEL
LIN {X 0,Y 9.094,Z 529.169,A -85,B 0,C 180,E1 -31719.525,E2 -31719.525} C_VEL
LIN {X 0,Y 6.45,Z 527.804,A -85,B 0,C 180,E1 -31770.12,E2 -31770.12} C_VEL
LIN {X 0,Y 11.871,Z 524.775,A -85,B 0,C 180,E1 -31832.772,E2 -31832.772} C_VEL
LIN {X 0,Y 19.64,Z 521.47,A -85,B 0,C 180,E1 -31847.239,E2 -31847.239} C_VEL
LIN {X 0,Y 24.614,Z 519.054,A -85,B 0,C 180,E1 -31852.581,E2 -31852.581} C_VEL
LIN {X 0,Y 29.36,Z 516.34,A -85,B 0,C 180,E1 -31857.477,E2 -31857.477} C_VEL
LIN {X 0,Y 38.54,Z 510.243,A -85,B 0,C 180,E1 -31865.419,E2 -31865.419} C_VEL
LIN {X 0,Y 44.598,Z 505.664,A -85,B 0,C 180,E1 -31869.061,E2 -31869.061} C_VEL
LIN {X 0,Y 43.806,Z 506.031,A -85,B 0,C 180,E1 -31875.657,E2 -31875.657} C_VEL
LIN {X 0,Y 42.447,Z 507.025,A -85,B 0,C 180,E1 -31877.76,E2 -31877.76} C_VEL
LIN {X 0,Y 31.447,Z 514.144,A -85,B 0,C 180,E1 -31878.153,E2 -31878.153} C_VEL
LIN {X 0,Y 18.474,Z 520.72,A -85,B 0,C 180,E1 -31877.864,E2 -31877.864} C_VEL
LIN {X 0,Y 7.241,Z 525.003,A -85,B 0,C 180,E1 -31873.486,E2 -31873.486} C_VEL
LIN {X 0,Y 7.157,Z 525.051,A -85,B 0,C 180,E1 -31870.31,E2 -31870.31} C_VEL
LIN {X 0,Y 18.23,Z 520.947,A -85,B 0,C 180,E1 -31868.343,E2 -31868.343} C_VEL
LIN {X 0,Y 28.404,Z 516.097,A -85,B 0,C 180,E1 -31868.033,E2 -31868.033} C_VEL
LIN {X 0,Y 39.05,Z 509.697,A -85,B 0,C 180,E1 -31868.035,E2 -31868.035} C_VEL
LIN {X 0,Y 42.6,Z 507.227,A -85,B 0,C 180,E1 -31868.051,E2 -31868.051} C_VEL
LIN {X 0,Y 44.598,Z 505.664,A -85,B 0,C 180,E1 -31869.061,E2 -31869.061} C_VEL
LIN {X 0,Y 47.589,Z 507.279,A -85,B 0,C 180,E1 -31870.405,E2 -31870.405} C_VEL
LIN {X 0,Y 47.589,Z 600,A -85,B 0,C 180,E1 -31870.405,E2 -31870.405} C_VEL
LIN {X 0,Y 47.589,Z 600,A -85,B 0,C 180,E1 -31870.405,E2 -31870.405}

QRS_NEXT_CUT()

QRS_NEXT()
QRS_HOME()

END
